{attribute 'qualified_only'}
{attribute 'strict'}
{attribute 'to_string'}
TYPE eCoolingSystemState :
(
	OFF 						:= 	0,
	EnclosureConditioning 		:= 	1,
	InverterStartup 			:= 	2,
	BatteryConditioning 		:= 	3,
	InverterPowerMode 			:= 	5,
	DeHum						:= 	4,
	DehumEnding					:= 	6,
	InverterConditioning		:=  7,
	EMSTOP						:=	10
)uint := OFF;
END_TYPE

(* stored: Version 1.1.0.1, ProductVersion 3.1.4024.12
   DUT eCoolingSystemState: Id {3d9938d8-59c8-4bba-9c8e-5ac8a873a19e} *)
